(* LS Electric XG5000 project: 통합 *)
(* PLC LSPLC *)

PROGRAM NewProgram (* task: 스캔 프로그램 *)
VAR
    T1 : TON;
    T2 : TON;
    근접센서1 AT %MX7 : BOOL;
    근접센서2 : BOOL;
    다음으로 : BOOL;
    대형1층동작 : TON;
    대형감지 AT %MX2 : BOOL;
    대형감지완료 AT %MX5 : BOOL;
    대형도착 AT %QX0.1.8 : BOOL;
    대형엘리도착 : BOOL;
    대형엘리동작1 : TON;
    대형입장 AT %IX0.0.2 : BOOL;
    도착 AT %QX0.1.13 : BOOL;
    레일동작 AT %QX0.1.4 : BOOL;
    레일정지 AT %QX0.1.5 : BOOL;
    물끓이기 : TON;
    물무게 : INT;
    물무게UDINT : UDINT;
    물무게곱하기 : INT;
    물투입 : TON;
    물투입시간 : TIME;
    물투입통과 : BOOL;
    섞기 : TON;
    섞기통과 : BOOL;
    소형감지 AT %MX0 : BOOL;
    소형감지완료 AT %MX3 : BOOL;
    소형도착 AT %QX0.1.6 : BOOL;
    소형입장 AT %IX0.0.0 : BOOL;
    시럽무게 : INT := 0;
    시럽무게UDINT : UDINT;
    시럽무게곱하기 : INT;
    시럽투입 : TON;
    시럽투입시간 : TIME;
    시럽투입여부 : BOOL;
    시럽투입통과 : BOOL;
    실링기계 : TON;
    실링기계동작 : BOOL;
    실링레일 : TON;
    실링레일동작 : BOOL;
    얼음선투입 AT %IX0.0.6 : BOOL;
    얼음선투입타이머 : TON;
    얼음선투입통과 : BOOL;
    얼음후투입 AT %IX0.0.7 : BOOL;
    얼음후투입타이머 : TON;
    얼음후투입통과 : BOOL;
    에이드투입 : BOOL := 0;
    엘리1층도착 : BOOL;
    엘리내려감 AT %QX0.1.11 : BOOL;
    엘리베이터대기 : TON;
    엘리베이터동작 AT %QX0.1.9 : BOOL;
    엘리베이터중지 AT %QX0.1.10 : BOOL;
    우유뎁히기 : TON;
    우유무게 : INT := 0;
    우유무게UDINT : UDINT;
    우유무게곱하기 : INT;
    우유투입 : TON;
    우유투입시간 : TIME;
    우유투입여부 : BOOL;
    우유투입통과 : BOOL;
    음료제조완료 AT %QX0.1.15 : BOOL;
    음료제조자가유지 : BOOL;
    음료주문 AT %IX0.0.5 : BOOL;
    일단멈춰 : BOOL := 0;
    일단멈춰2 : BOOL;
    일단멈춰3 : BOOL;
    자동차입장감지센서 AT %QX0.1.0 : BOOL;
    자동차퇴장감지 AT %IX0.0.4 : BOOL;
    자동차퇴장알림 AT %QX0.1.12 : BOOL;
    주차차단기개방 AT %QX0.1.1 : BOOL;
    주차차단기차단 : BOOL;
    중형1층동작 : TON;
    중형감지 AT %MX1 : BOOL;
    중형감지완료 AT %MX4 : BOOL;
    중형도착 AT %QX0.1.7 : BOOL;
    중형엘리도착 : BOOL;
    중형엘리동작1 : TON;
    중형입장 AT %IX0.0.1 : BOOL;
    지나감감지 : TON;
    커피무게 : INT;
    커피무게UDINT : UDINT;
    커피무게곱하기 : INT;
    커피배달중 AT %QX0.1.14 : BOOL;
    커피제작시작 AT %QX0.1.2 : BOOL;
    커피제작완료 AT %QX0.1.3 : BOOL;
    커피주문 AT %IX0.0.3 : BOOL;
    커피주문완료 AT %MX6 : BOOL;
    커피추출 : TON;
    커피투입 : TON;
    커피투입시간 : TIME;
    커피투입시작 : BOOL;
    커피투입통과 : BOOL;
    퇴장알림 : TON;
END_VAR
VAR
    _t1 : BOOL;
    _t2 : BOOL;
END_VAR

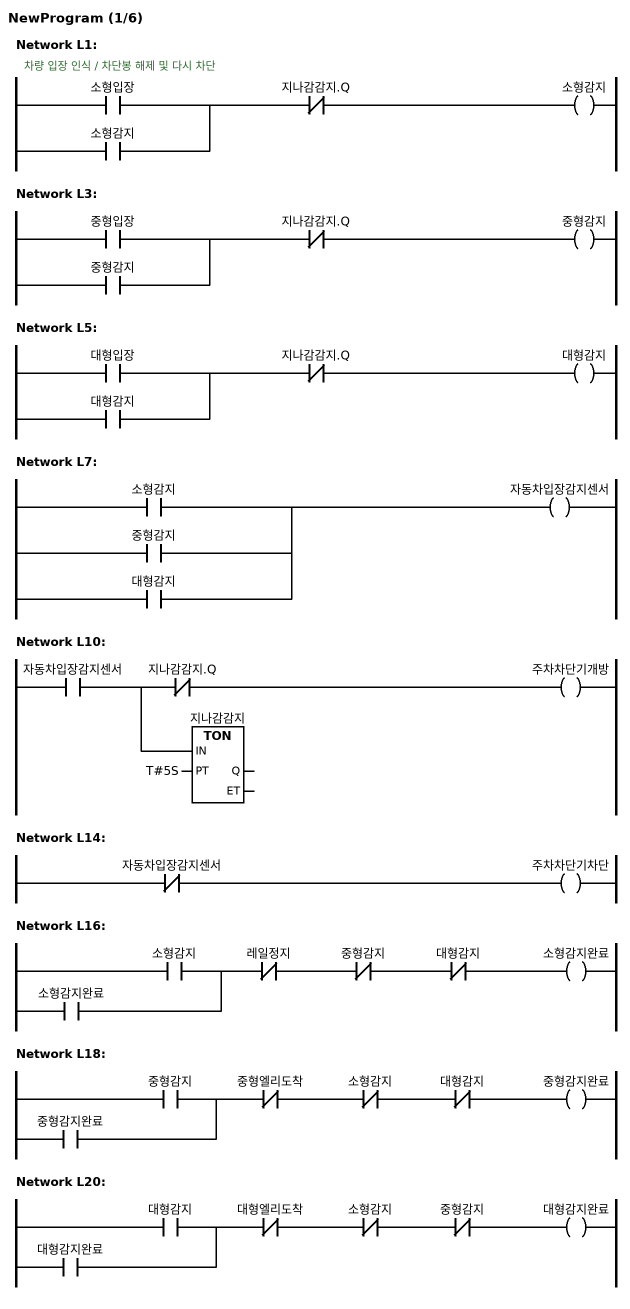
(* 차량 입장 인식 / 차단봉 해제 및 다시 차단 *)
(* Rung L1 *)
소형감지 := (소형입장 OR 소형감지) AND NOT 지나감감지.Q;
(* Rung L3 *)
중형감지 := (중형입장 OR 중형감지) AND NOT 지나감감지.Q;
(* Rung L5 *)
대형감지 := (대형입장 OR 대형감지) AND NOT 지나감감지.Q;
(* Rung L7 *)
자동차입장감지센서 := 소형감지 OR 중형감지 OR 대형감지;
(* Rung L10 *)
주차차단기개방 := 자동차입장감지센서 AND NOT 지나감감지.Q;
지나감감지(IN := 자동차입장감지센서, PT := T#5S);
(* Rung L14 *)
주차차단기차단 := NOT 자동차입장감지센서;
(* Rung L16 *)
소형감지완료 := (소형감지 OR 소형감지완료) AND NOT 레일정지 AND NOT 중형감지 AND NOT 대형감지;
(* Rung L18 *)
중형감지완료 := (중형감지 OR 중형감지완료) AND NOT 중형엘리도착 AND NOT 소형감지 AND NOT 대형감지;
(* Rung L20 *)
대형감지완료 := (대형감지 OR 대형감지완료) AND NOT 대형엘리도착 AND NOT 소형감지 AND NOT 중형감지;

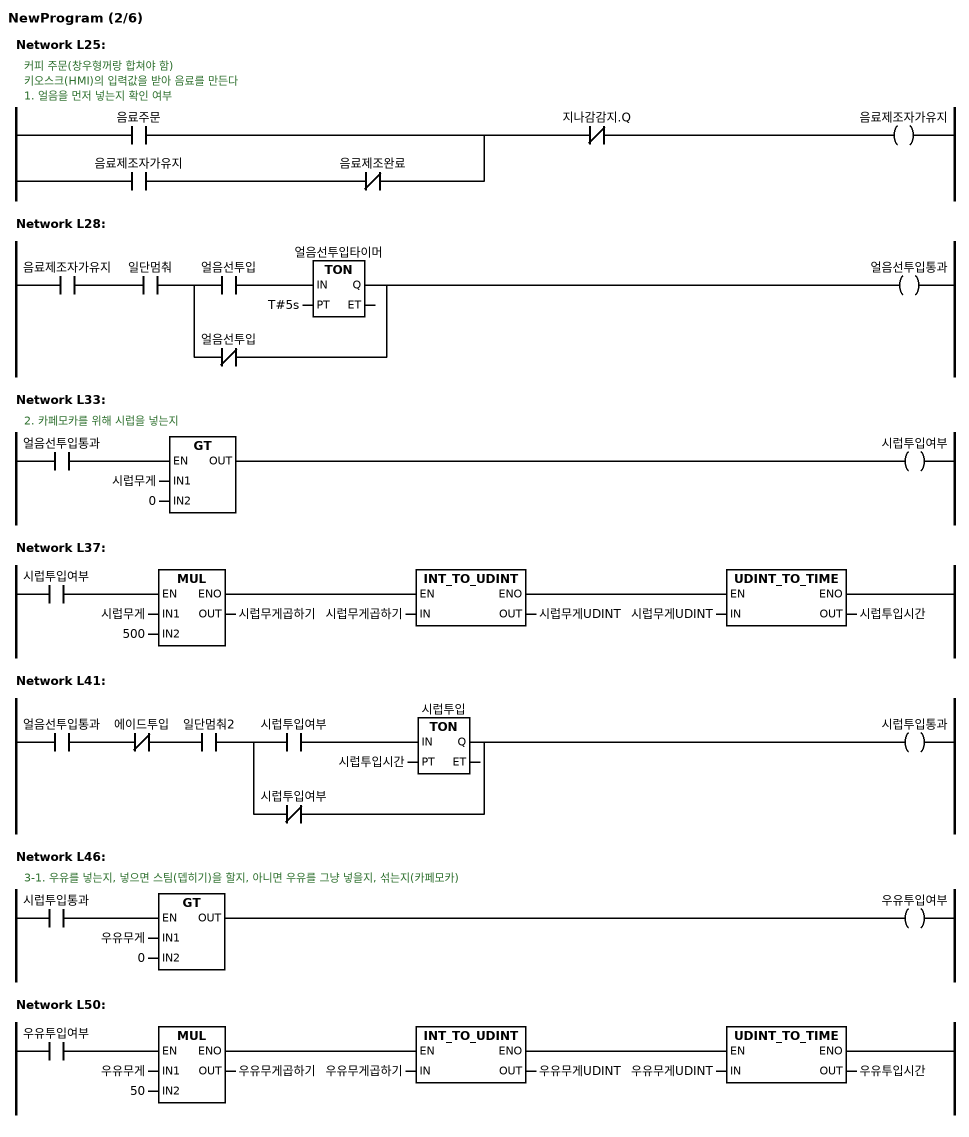
(* 커피 주문(창우형꺼랑 합쳐야 함) *)
(* 키오스크(HMI)의 입력값을 받아 음료를 만든다 *)
(* 1. 얼음을 먼저 넣는지 확인 여부 *)
(* Rung L25 *)
음료제조자가유지 := (음료주문 OR (음료제조자가유지 AND NOT 음료제조완료)) AND NOT 지나감감지.Q;
(* Rung L28 *)
얼음선투입타이머(IN := 음료제조자가유지 AND 일단멈춰 AND 얼음선투입, PT := T#5s);
얼음선투입통과 := 얼음선투입타이머.Q OR (음료제조자가유지 AND 일단멈춰 AND NOT 얼음선투입);
(* 2. 카페모카를 위해 시럽을 넣는지 *)
(* Rung L33 *)
IF 얼음선투입통과 THEN _t1 := 시럽무게 > 0; END_IF;
시럽투입여부 := _t1;
(* Rung L37 *)
IF 시럽투입여부 THEN
    시럽무게곱하기 := 시럽무게 * 500;
    시럽무게UDINT := INT_TO_UDINT(시럽무게곱하기);
    시럽투입시간 := UDINT_TO_TIME(시럽무게UDINT);
END_IF;
(* Rung L41 *)
시럽투입(IN := 얼음선투입통과 AND NOT 에이드투입 AND 일단멈춰2 AND 시럽투입여부, PT := 시럽투입시간);
시럽투입통과 := 시럽투입.Q OR (얼음선투입통과 AND NOT 에이드투입 AND 일단멈춰2 AND NOT 시럽투입여부);
(* 3-1. 우유를 넣는지, 넣으면 스팀(뎁히기)을 할지, 아니면 우유를 그냥 넣을지, 섞는지(카페모카) *)
(* Rung L46 *)
IF 시럽투입통과 THEN _t2 := 우유무게 > 0; END_IF;
우유투입여부 := _t2;
(* Rung L50 *)
IF 우유투입여부 THEN
    우유무게곱하기 := 우유무게 * 50;
    우유무게UDINT := INT_TO_UDINT(우유무게곱하기);
    우유투입시간 := UDINT_TO_TIME(우유무게UDINT);
END_IF;

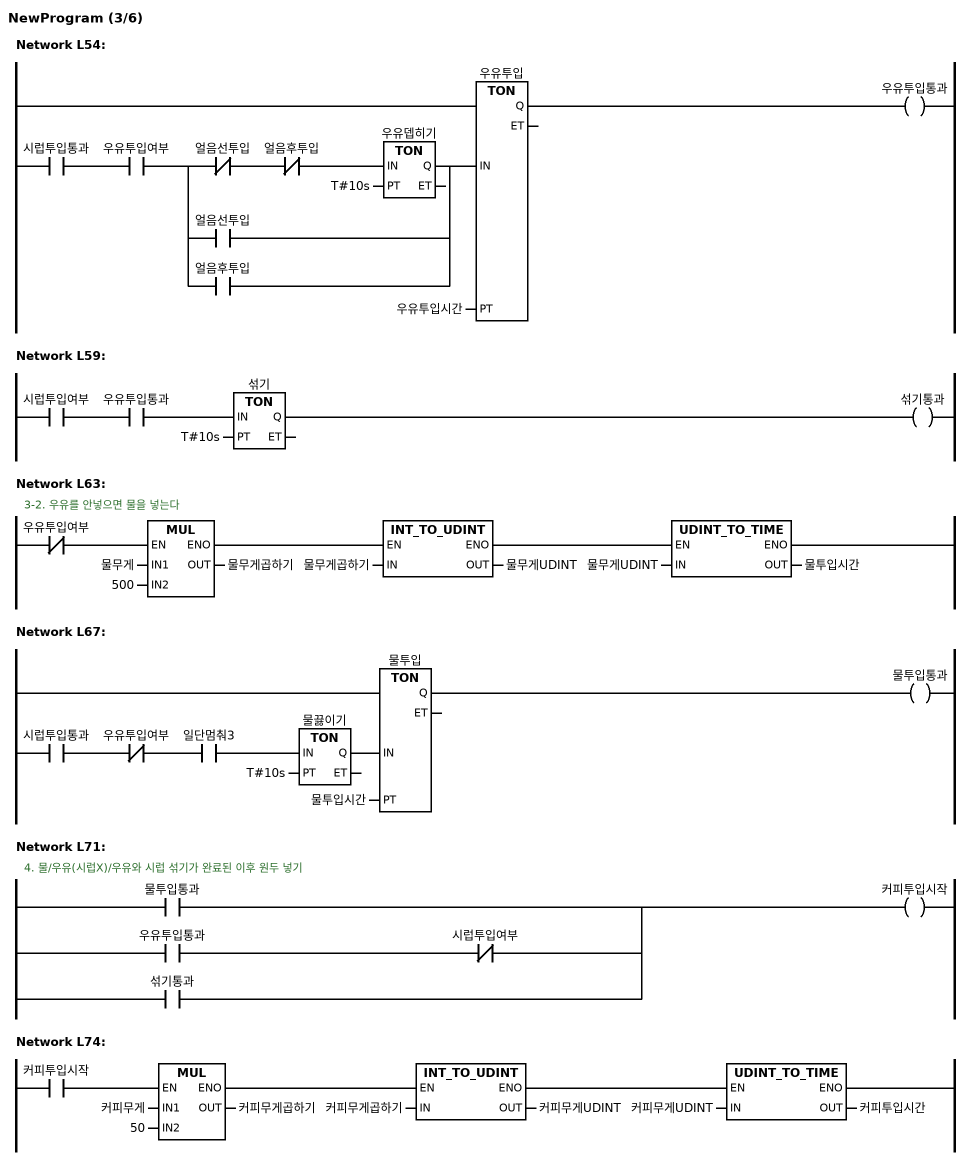
(* Rung L54 *)
우유뎁히기(IN := 시럽투입통과 AND 우유투입여부 AND NOT 얼음선투입 AND NOT 얼음후투입, PT := T#10s);
우유투입(IN := 우유뎁히기.Q OR (시럽투입통과 AND 우유투입여부 AND (얼음선투입 OR 얼음후투입)), PT := 우유투입시간);
우유투입통과 := 우유투입.Q;
(* Rung L59 *)
섞기(IN := 시럽투입여부 AND 우유투입통과, PT := T#10s);
섞기통과 := 섞기.Q;
(* 3-2. 우유를 안넣으면 물을 넣는다 *)
(* Rung L63 *)
IF NOT 우유투입여부 THEN
    물무게곱하기 := 물무게 * 500;
    물무게UDINT := INT_TO_UDINT(물무게곱하기);
    물투입시간 := UDINT_TO_TIME(물무게UDINT);
END_IF;
(* Rung L67 *)
물끓이기(IN := 시럽투입통과 AND NOT 우유투입여부 AND 일단멈춰3, PT := T#10s);
물투입(IN := 물끓이기.Q, PT := 물투입시간);
물투입통과 := 물투입.Q;
(* 4. 물/우유(시럽X)/우유와 시럽 섞기가 완료된 이후 원두 넣기 *)
(* Rung L71 *)
커피투입시작 := 물투입통과 OR (우유투입통과 AND NOT 시럽투입여부) OR 섞기통과;
(* Rung L74 *)
IF 커피투입시작 THEN
    커피무게곱하기 := 커피무게 * 50;
    커피무게UDINT := INT_TO_UDINT(커피무게곱하기);
    커피투입시간 := UDINT_TO_TIME(커피무게UDINT);
END_IF;

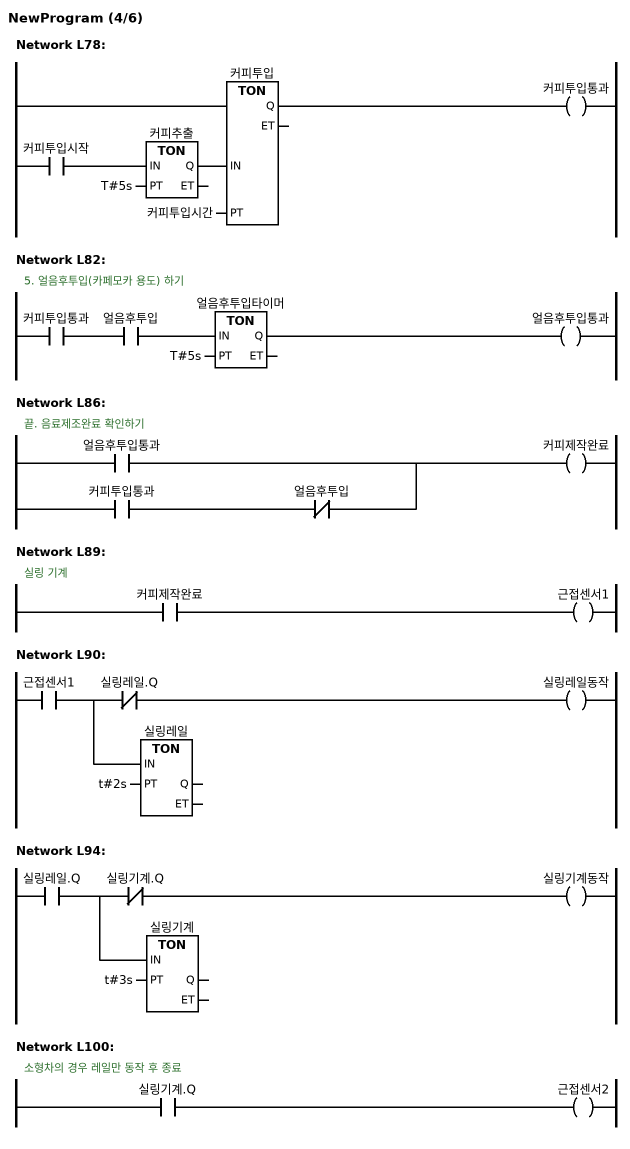
(* Rung L78 *)
커피추출(IN := 커피투입시작, PT := T#5s);
커피투입(IN := 커피추출.Q, PT := 커피투입시간);
커피투입통과 := 커피투입.Q;
(* 5. 얼음후투입(카페모카 용도) 하기 *)
(* Rung L82 *)
얼음후투입타이머(IN := 커피투입통과 AND 얼음후투입, PT := T#5s);
얼음후투입통과 := 얼음후투입타이머.Q;
(* 끝. 음료제조완료 확인하기 *)
(* Rung L86 *)
커피제작완료 := 얼음후투입통과 OR (커피투입통과 AND NOT 얼음후투입);
(* 실링 기계 *)
(* Rung L89 *)
근접센서1 := 커피제작완료;
(* Rung L90 *)
실링레일동작 := 근접센서1 AND NOT 실링레일.Q;
실링레일(IN := 근접센서1, PT := t#2s);
(* Rung L94 *)
실링기계동작 := 실링레일.Q AND NOT 실링기계.Q;
실링기계(IN := 실링레일.Q, PT := t#3s);
(* 소형차의 경우 레일만 동작 후 종료 *)
(* Rung L100 *)
근접센서2 := 실링기계.Q;

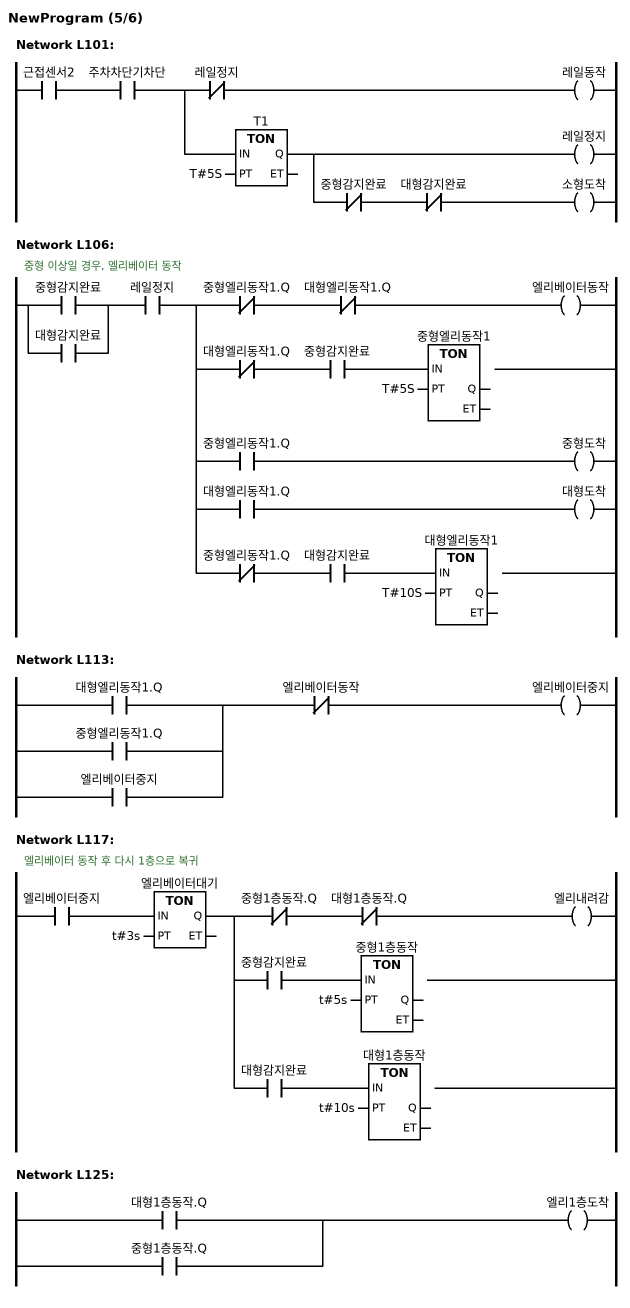
(* Rung L101 *)
레일동작 := 근접센서2 AND 주차차단기차단 AND NOT 레일정지;
T1(IN := 근접센서2 AND 주차차단기차단, PT := T#5S);
레일정지 := T1.Q;
소형도착 := T1.Q AND NOT 중형감지완료 AND NOT 대형감지완료;
(* 중형 이상일 경우, 엘리베이터 동작 *)
(* Rung L106 *)
엘리베이터동작 := (중형감지완료 OR 대형감지완료) AND 레일정지 AND NOT 중형엘리동작1.Q AND NOT 대형엘리동작1.Q;
중형엘리동작1(IN := (중형감지완료 OR 대형감지완료) AND 레일정지 AND NOT 대형엘리동작1.Q AND 중형감지완료, PT := T#5S);
중형도착 := (중형감지완료 OR 대형감지완료) AND 레일정지 AND 중형엘리동작1.Q;
대형도착 := (중형감지완료 OR 대형감지완료) AND 레일정지 AND 대형엘리동작1.Q;
대형엘리동작1(IN := (중형감지완료 OR 대형감지완료) AND 레일정지 AND NOT 중형엘리동작1.Q AND 대형감지완료, PT := T#10S);
(* Rung L113 *)
엘리베이터중지 := (대형엘리동작1.Q OR 중형엘리동작1.Q OR 엘리베이터중지) AND NOT 엘리베이터동작;
(* 엘리베이터 동작 후 다시 1층으로 복귀 *)
(* Rung L117 *)
엘리베이터대기(IN := 엘리베이터중지, PT := t#3s);
엘리내려감 := 엘리베이터대기.Q AND NOT 중형1층동작.Q AND NOT 대형1층동작.Q;
중형1층동작(IN := 엘리베이터대기.Q AND 중형감지완료, PT := t#5s);
대형1층동작(IN := 엘리베이터대기.Q AND 대형감지완료, PT := t#10s);
(* Rung L125 *)
엘리1층도착 := 대형1층동작.Q OR 중형1층동작.Q;

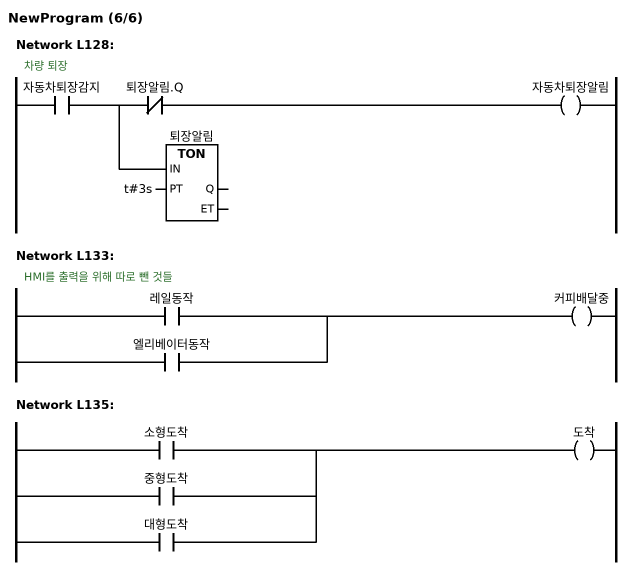
(* 차량 퇴장 *)
(* Rung L128 *)
자동차퇴장알림 := 자동차퇴장감지 AND NOT 퇴장알림.Q;
퇴장알림(IN := 자동차퇴장감지, PT := t#3s);
(* HMI를 출력을 위해 따로 뺀 것들 *)
(* Rung L133 *)
커피배달중 := 레일동작 OR 엘리베이터동작;
(* Rung L135 *)
도착 := 소형도착 OR 중형도착 OR 대형도착;
END_PROGRAM